// TIA Portal V17 export
// export: Created 2025-06-20T13:04:35.3999496Z, ExportSetting WithDefaults, DisplayName Totally Integrated Automation Portal, DisplayVersion V17 Update 8, DisplayName TIA Portal Openness, DisplayVersion V17 Update 8, DisplayName TIA Portal Version Control Interface, DisplayVersion V17, DisplayName SINAMICS Startdrive Advanced, DisplayVersion V17 SP2, DisplayName SINAMICS Startdrive G110M, G120, G120C, G120D, G120P, G115D, DisplayVersion V17 SP2, DisplayName SINAMICS Startdrive G130, G150, S120, S150, SINAMICS MV, S210, DisplayVersion V17 SP2, DisplayName STEP 7 Professional, DisplayVersion V17 Update 8, DisplayName SINUMERIK ONE STEP 7 Toolbox, DisplayVersion V17 Update 12, DisplayName SINUMERIK ONE PLC Basic Program Plus, DisplayVersion V17 Update 12, DisplayName SINUMERIK 840D sl STEP 7 Toolbox, DisplayVersion V17 Update 12, DisplayName STEP 7 Safety, DisplayVersion V17 Update 6, DisplayName WinCC Advanced, DisplayVersion V17 Update 8
DATA_BLOCK "DB16468_U3_MEAS_RECONNECT_N"   // DB16468
{ DB_Accessible_From_OPC_UA := 'FALSE' }
VERSION : 0.1
// stored: AutoNumber false, DBAccessibleFromOPCUA false, DBAccessibleFromWebserver true, InstanceOfName FB16001_METHODS_CONNECTION_MGR, InstanceOfType FB
"FB16001_METHODS_CONNECTION_MGR"
   // VAR_INPUT
   //    CONNECTION_BLOCK_DONE : Bool;
   //    CONNECTION_BLOCK_ERROR : Bool;
   //    CONNECTION_BLOCK_BUSY : Bool;
   //    READ_VARIABLES_BLOCK_ERROR : Bool;
   //    DISCONNECT_BLOCK_DONE : Bool;
   //    DISCONNECT_BLOCK_BUSY : Bool;
   //    RESET_CONNECTION_ATTEMPTS : Bool;
   //    OPC_UA_CONNECT_STATUS : DWord;
   //    OPC_UA_GET_INDEX_LIST_STATUS : DWord;
   //    OPC_UA_GET_HANDLE_LIST_STATUS : DWord;
   //    OPC_UA_GET_METHOD_LIST_STATUS : DWord;
   //    OPC_UA_GET_METHOD_LIST_STATUS_1 : DWord;
   //    OPC_UA_RELEASE_HANDLE_LIST_STATUS : DWord;
   //    OPC_UA_RELEASE_METHOD_LIST_STATUS : DWord;
   //    OPC_UA_RELEASE_METHOD_LIST_STATUS_1 : DWord;
   //    OPC_UA_READ_VARIABLES_STATUS : DWord;
   //    OPC_UA_DISCONNECT_STATUS : DWord;
   //    OPC_UA_CONNECTION_GET_STATUS : DWord;
   //    MAX_CON_ATTEMPTS : Int;
   // END_VAR
   // VAR_OUTPUT
   //    RETRY_CONNECTION : Bool;
   //    DISCONNECT : Bool;
   //    CONNECTION_ERROR : Bool;
   //    CONNECTION_ERROR_STATUS : "CONNECTION_ERROR_STATUS";
   // END_VAR
   // VAR
   //    CONNECTION_ERROR_MEM : Bool;
   //    CONNECTION_DONE_MEM : Bool;
   //    DISCONNECT_DONE_MEM : Bool;
   //    ERROR_COUNTER : Int;
   //    AUX_PULSE : Bool;
   //    AUX_PULSE_1 : Bool;
   //    AUX_PULSE_2 : Bool;
   //    LAST_ERROR_TIME_STAMP : DTL;
   //    RET_VAL : Int;
   // END_VAR
BEGIN
END_DATA_BLOCK
